FUNCTION_BLOCK FB_Klep IMPLEMENTS ITF_UnitKlep
VAR
    _cmdOpen : BOOL;   // laatst aangevraagde command
    _status  : BOOL;   // huidige status van de klep
END_VAR

PROPERTY PUBLIC Status : BOOL
GET
Status := _status;   // status uitlezen
END_GET
SET
END_SET
END_PROPERTY

METHOD PUBLIC SturingOpen : BOOL
VAR_INPUT
	i_bOpen	: BOOL; // TRUE = open, FALSE = dicht
END_VAR
_cmdOpen := i_bOpen;
_status  := _cmdOpen;
END_METHOD

END_FUNCTION_BLOCK

(* stored: Version 1.1.0.1
   POU FB_Klep: Id {a42b2b1d-3d0d-4ad8-8a49-e659df0386f5}, SpecialFunc None
   Folder Methods: Id {215c97dc-4785-4f3f-80d3-672f5b9c53d7}
   Folder Properties: Id {8948e215-6589-49b0-8016-a5dec4d22119}
   Property Status: Id {fac60b85-9052-4a73-9fa5-0cc4b71f46f0}
   Get Get: Id {126ac777-00b4-45e9-900d-48260272a880}
   Set Set: Id {52aaba85-13ed-4e62-a0db-c488bafb88d7}
   Method SturingOpen: Id {789bb220-7b95-473c-9a9f-a5eb352b7b20} *)
